PROGRAM PRG_90_GeneralConditions
VAR
END_VAR

(* Errors Cabinet *)
Errors_Cabinet.ERRORS[0].0 := NOT IN_bSawMOLReady ;		// Saw blade motor overload
//Errors_Cabinet.ERRORS[0].1 := NOT IN_bCableReelMOLReady ;		// Cable reel motor overload
//Errors_Cabinet.ERRORS[0].2 := NOT IN_bHoseReelMOLReady ;		// Hose reel motor overload

(* Errors TwinSAFE *)
Errors_TwinSAFE.ERRORS[0].0 := bEstopPanelErr ;		// E-stop control panel
Errors_TwinSAFE.ERRORS[0].1 := bEstopLeftErr ;		// E-stop left side
Errors_TwinSAFE.ERRORS[0].2 := bEstopRightErr ;		// E-stop right side

(* Warnings Saw *)
Warnings_Saw.ERRORS[0].0 := NOT bAllowCarriageMovement ;		// Carriage movement not allowed
Warnings_Saw.ERRORS[0].1 := NOT bAllowTurretMovement ;		// Turret movement not allowed
Warnings_Saw.ERRORS[0].2 := PRG_11_ScreenButtons.SR_CarriageEnableTimeout.Q1 ;		// Carriage enable button timed out
Warnings_Saw.ERRORS[0].3 := PRG_11_ScreenButtons.SR_TurretEnableTimeout.Q1 ;		// Turret enable button timed out
Warnings_Saw.ERRORS[0].4 := PRG_11_ScreenButtons.SR_DriveFastTimeout.Q1 ;		// Drive fast button timed out
Warnings_Saw.ERRORS[0].5 := NOT bDriveAllowed ;		// X-Drive not allowed
Warnings_Saw.ERRORS[0].6 := NOT (OUT_bSawON AND bTurret045Range AND bCarriageCentreRef) ;		// Auto CrossCut not ready
Warnings_Saw.ERRORS[0].7 := NOT OUT_bSawON AND NOT bSawUpLimit ;		// Saw blade not ready to turn on
Warnings_Saw.ERRORS[0].8 := FALSE ;

(* Errors Axes *)
Errors_Axes.ERRORS[0].0 := fbCarriage_manager.Error ;		// Carriage axis manager error
Errors_Axes.ERRORS[0].1 := fbCrossCut_manager.Error ;		// CrossCut axis manager error
Errors_Axes.ERRORS[0].2 := fbTurret_manager.Error ;		// Turret axis manager error
Errors_Axes.ERRORS[0].3 := fbXDrive_manager.Error ;		// X-Drive axis manager error
Errors_Axes.ERRORS[0].4 := fbZ1_manager.Error ;		// Z1 (panel side) axis manager error
Errors_Axes.ERRORS[0].5 := fbZ2_manager.Error ;		// Z2 (reel side) axis manager error

(* Errors Auto CrossCut time out *)
Errors_AutoCrossCut.ERRORS[0].0 := 	PRG_08_AutoCrossCut.SR_WatchdogTriggered.Q1
								AND PRG_08_AutoCrossCut.iStepErr = 20 ;
Errors_AutoCrossCut.ERRORS[0].1 := 	PRG_08_AutoCrossCut.SR_WatchdogTriggered.Q1
								AND PRG_08_AutoCrossCut.iStepErr = 30 ;
Errors_AutoCrossCut.ERRORS[0].2 := 	PRG_08_AutoCrossCut.SR_WatchdogTriggered.Q1
								AND PRG_08_AutoCrossCut.iStepErr = 40 ;
Errors_AutoCrossCut.ERRORS[0].3 := 	PRG_08_AutoCrossCut.SR_WatchdogTriggered.Q1
								AND PRG_08_AutoCrossCut.iStepErr = 50 ;
Errors_AutoCrossCut.ERRORS[0].4 := 	PRG_08_AutoCrossCut.SR_WatchdogTriggered.Q1
								AND PRG_08_AutoCrossCut.iStepErr = 60 ;
								
(* Errors Lifting Position time out *)
Errors_LiftingPosition.ERRORS[0].0 := 	PRG_09_HomePosition.SR_WatchdogTriggered.Q1
									AND PRG_09_HomePosition.iStepErr = 10 ;
Errors_LiftingPosition.ERRORS[0].1 := 	PRG_09_HomePosition.SR_WatchdogTriggered.Q1
									AND PRG_09_HomePosition.iStepErr = 20 ;
Errors_LiftingPosition.ERRORS[0].2 := 	PRG_09_HomePosition.SR_WatchdogTriggered.Q1
									AND PRG_09_HomePosition.iStepErr = 30 ;
Errors_LiftingPosition.ERRORS[0].3 := 	PRG_09_HomePosition.SR_WatchdogTriggered.Q1
									AND PRG_09_HomePosition.iStepErr = 40 ;
Errors_LiftingPosition.ERRORS[0].4 := 	PRG_09_HomePosition.SR_WatchdogTriggered.Q1
									AND PRG_09_HomePosition.iStepErr = 50 ;
								
(* Errors CrossCut Position time out *)
Errors_CrossCutPosition.ERRORS[0].0 := 	PRG_10_CrossCutPosition.SR_WatchdogTriggered.Q1
									AND PRG_10_CrossCutPosition.iStepErr = 10 ;
Errors_CrossCutPosition.ERRORS[0].1 := 	PRG_10_CrossCutPosition.SR_WatchdogTriggered.Q1
									AND PRG_10_CrossCutPosition.iStepErr = 20 ;
Errors_CrossCutPosition.ERRORS[0].2 := 	PRG_10_CrossCutPosition.SR_WatchdogTriggered.Q1
									AND PRG_10_CrossCutPosition.iStepErr = 30 ;
Errors_CrossCutPosition.ERRORS[0].3 := 	PRG_10_CrossCutPosition.SR_WatchdogTriggered.Q1
									AND PRG_10_CrossCutPosition.iStepErr = 40 ;

END_PROGRAM

(* stored: Version 1.1.0.1, ProductVersion 3.1.4024.15
   POU PRG_90_GeneralConditions: Id {b8d55638-6e09-4e51-9ff3-9cbb2bc10f26}, SpecialFunc None *)
